TYPE ST_Input_breakersettings :
STRUCT
	AutoConnect				: BOOL;
	ShutdownDisconnect		: BOOL;
	EMstopDisconnect		: BOOL;
	CurrentLimitDisconnect 	: BOOL;
	CurrentLimitRetries		: BYTE;
END_STRUCT
END_TYPE

(* stored: Version 1.1.0.1, ProductVersion 3.1.4026.18
   DUT ST_Input_breakersettings: Id {77f5aa65-782b-46da-b43a-d70ab593c6c8} *)
